// TIA Portal V20 export
FUNCTION_BLOCK "FB - Machine Modules"   // FB1, LAD
TITLE = Machine - Modules
{ S7_Optimized_Access := 'TRUE' }
// stored: MemoryReserve 100, SetENOAutomatically false
BEGIN

REGION Network 1: StateHandler process 1 - table
END_REGION

REGION Network 2: StateHandler process 2 - table
END_REGION
END_FUNCTION_BLOCK
